PROGRAM ControlParameters
VAR
END_VAR

END_PROGRAM

(* stored: Version 1.1.0.1, ProductVersion 3.1.4024.9
   POU ControlParameters: Id {ffc61bee-c1b2-401b-8834-f726b798ade9}, SpecialFunc None *)
